// TIA Portal V20 export
TYPE "LKinCtrl_typeFlagBufferElement"
   STRUCT
      pathDataName : String["LKINCTRL_LENGTH_OF_PATHDATA_NAME"] := '';   // PathData name of specific command
      pathDataIdentifier : DInt;   // PathData identifier counter of specific command
      cmdId : DInt := 0;   // cmdId of command in PathData
      isIntermediateCmd : Bool;   // TRUE: command is intermediate command
      setFlags : Array[1.."LKINCTRL_NO_OF_CMD_SETFLAGS"] of "LKinCtrl_typeSetFlagElement_Bool";   // setFlags structure equal to PathData command entry
      valueFlags : Array[1.."LKINCTRL_NO_OF_CMD_VALUEFLAGS"] of "LKinCtrl_typeSetFlagElement_LReal";   // setFlags structure equal to PathData command entry
   END_STRUCT;
END_TYPE
